TYPE DUT_HMI_12_MANUALS :
STRUCT
	PS : ARRAY[0..CNC.NUM_MAX_MANUALS_12-1] OF BOOL;
	LS : ARRAY[0..CNC.NUM_MAX_MANUALS_12-1] OF BOOL;
END_STRUCT
END_TYPE

(* stored: Version 1.1.0.1, ProductVersion 3.1.4024.13
   DUT DUT_HMI_12_MANUALS: Id {ef229bed-f8fd-4ba1-89ee-cfc01ced473d} *)
